FUNCTION strlen : UINT
VAR_INPUT
	pStr	: POINTER TO STRING;
END_VAR
VAR
	tmpStrLen	: UINT;
	pArr		: POINTER TO BYTE;
END_VAR

(********************************************************************
 * COPYRIGHT -- Hewlett-Packard Company
 ********************************************************************
 * Program: logLib
 * File: logLib.st
 * Author: 
 * Created: Feb 20, 2017
 ********************************************************************
 * Implementation of program logLib
 ********************************************************************) 

tmpStrLen	:= 0;
pArr		:= pStr;
WHILE pArr^ <> 0 DO
	tmpStrLen	:= tmpStrLen + 1;
	pArr	:= pArr + 1;
END_WHILE
strlen	:= tmpStrLen;
RETURN;

END_FUNCTION

(* stored: Version 1.1.0.1, ProductVersion 3.1.4024.3
   POU strlen: Id {24503334-8e3c-07aa-1523-3ce3e40abeca}, SpecialFunc None *)
